# EPICS autosave request: smc/smc_settings.req
$(P):LIM:FIELD:NOW
$(P):STS:MAGMODE
